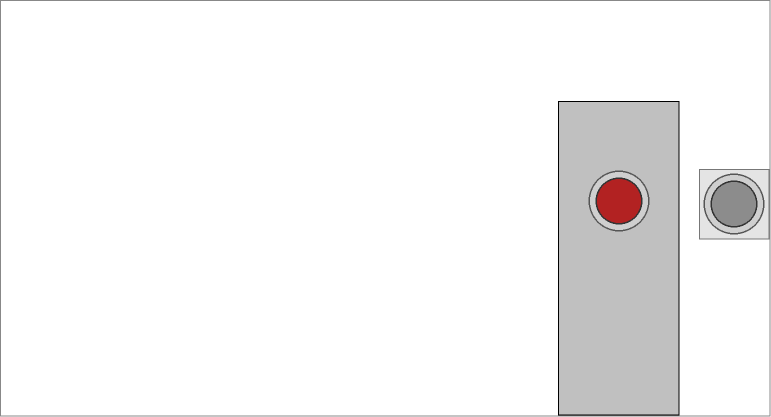
VISUALIZATION FakeButtons  // 771x417
    Rectangle (558,101 121x314)
    Lamp1 (584,166 70x70), style: Lamp-Lamp1-Red
    PushSwitchLed (699,169 70x70), behaviour: TOGGLE, style: Switch-PushSwitchLed-Gray
END_VISUALIZATION

(* stored: Version 1.1.0.1, ProductVersion 3.1.0.36
   Visu FakeButtons: Id {212326d2-d590-4aeb-800c-70dc996e0b55} *)
